// Mitsubishi GX Works2 project: 인칭이동량   PLC: Q02/Q02H

PROGRAM MAIN
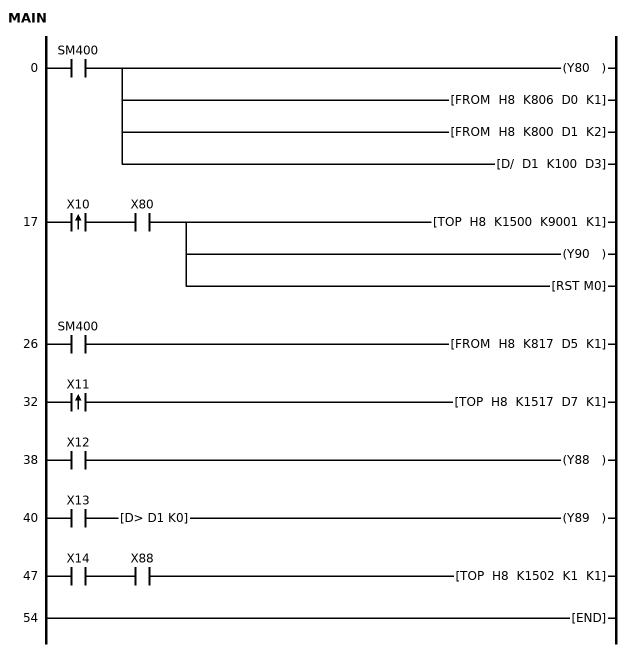
0     LD      SM400
      OUT     Y80
      FROM    H8 K806 D0 K1
      FROM    H8 K800 D1 K2
      D/      D1 K100 D3
17    LDP     X10
      AND     X80
      TOP     H8 K1500 K9001 K1
      OUT     Y90
      RST     M0
26    LD      SM400
      FROM    H8 K817 D5 K1
32    LDP     X11
      TOP     H8 K1517 D7 K1
38    LD      X12
      OUT     Y88
40    LD      X13
      ANDD>   D1 K0
      OUT     Y89
47    LD      X14
      AND     X88
      TOP     H8 K1502 K1 K1
54    END
END_PROGRAM
